PROGRAM MAIN
VAR
    bStartupDone   : BOOL := FALSE;   // runs once on boot
    tonStartDelay  : TON;             // small delay to let DALI bus settle first
END_VAR


POU();
WallLight_POU();

END_PROGRAM

(* stored: Version 1.1.0.1, ProductVersion 3.1.4024.16
   POU MAIN: Id {7d680b2f-8db9-4f1e-8602-1c7527d7b88c}, SpecialFunc None *)
